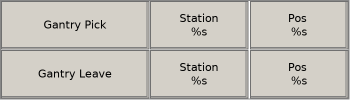
VISUALIZATION _VisuGantryPickLeave  // 350x100
    Button (1,1 148x48), "Gantry Pick"
        toggle ComGVL._fbTryOutGantryPickEn
    Button (1,50 148x48), "Gantry Leave"
        toggle ComGVL._fbTryOutGantryLeaveEn
    Button (150,1 98x48), "Station %s", text variable: ComGVL._fbTryOutGantryPickStation
        OnMouseDown: write the text variable via VisuDialogs.Numpad, min 1, max 4, title 'Station'
    Button (150,50 98x48), "Station %s", text variable: ComGVL._fbTryOutGantryLeaveStation
        OnMouseDown: write the text variable via VisuDialogs.Numpad, min 1, max 4, title 'Station'
    Button (250,1 98x48), "Pos %s", text variable: ComGVL._fbTryOutGantryPickPos
        OnMouseDown: write the text variable via VisuDialogs.Numpad, min 1, max 9, title 'Position'
    Button (250,50 98x48), "Pos %s", text variable: ComGVL._fbTryOutGantryLeavePos
        OnMouseDown: write the text variable via VisuDialogs.Numpad, min 1, max 9, title 'Position'
END_VISUALIZATION

(* stored: Version 1.1.0.1, ProductVersion 3.1.4024.2
   Visu _VisuGantryPickLeave: Id {37b71458-e639-4855-a0f2-a6b663cf5cea} *)
